// TIA Portal V20 export
TYPE "UDT_MTP_BinVlv"
TITLE = MTPDataObjectSUCLibrary/DataAssembly/BinVlv
   STRUCT
      CloseOp : Bool := FALSE;   // Close command from Operator (relevant, if StateOpAct) 0-->1:request from POL 1-->0 acknowledge from PEA(see Handshake)
      OpenOp : Bool := FALSE;   // Open command from Operator (relevant, if StateOpAct) 0-->1:request from POL 1-->0 acknowledge from PEA(see Handshake)
      OSLevel : Byte := 16#00;   // OSLevel variable
      StateChannel { ExternalWritable := 'False'} : Bool;   // Selection of the active Operation Mode interaction channel 0: the operator switches (*Op) shall be used 1: the automatic switches (*Aut) shall be used
      StateOffAut { ExternalWritable := 'False'} : Bool;   // Set OperationMode to Offline by automatic interaction (relevant, if StateChannel) 1:OperationMode is set to Offline 0:no operation
      StateOffOp : Bool;   // Set OperationMode to Offline by operator interaction (relevant, if not StateChannel) 0-->1:request to set OperationMode to Offline 1-->0:acknowledge by PEA
      StateOpAut { ExternalWritable := 'False'} : Bool;   // Set OperationMode to Operator by automatic interaction (relevant, if StateChannel) 1:OperationMode is set to Manual 0:no operation
      StateOpOp : Bool;   // Set OperationMode to Operator by operator interaction (relevant, if not StateChannel) 0-->1:request to set OperationMode to Manual 1-->0:acknowledge by PEA
      StateAutAut { ExternalWritable := 'False'} : Bool;   // Set OperationMode to Automatic by automatic interaction (relevant, if StateChannel) 1:OperationMode is set to Automatic 0:no operation
      StateAutOp : Bool;   // Set OperationMode to Automatic by operator interaction (relevant, if not StateChannel) 0-->1:request to set OperationMode is to Automatic 1-->0:acknowledge by PEA
      StateOpAct { ExternalWritable := 'False'} : Bool;   // 1: current mode is Operator 0: current mode is not Operator
      StateAutAct { ExternalWritable := 'False'} : Bool;   // 1: current mode is Automatic 0: current mode is not Automatic
      StateOffAct { ExternalWritable := 'False'} : Bool;   // 1: current mode is Offline 0: current mode is not Offline
      CSF { ExternalWritable := 'False'} : Bool;   // Reserved
      WQC { ExternalWritable := 'False'} : Byte := 16#FF;   // Worst Quality code
      CloseAut { ExternalWritable := 'False'} : Bool := FALSE;   // Set Valve to Close by Automatic (relevant, if StateAutAct) 1:close request 0:no close request
      OpenAut { ExternalWritable := 'False'} : Bool := FALSE;   // Set Valve to Open by Automatic (relevant, if StateAutAct) 1:open request 0:no open request
      Ctrl { ExternalWritable := 'False'} : Bool := FALSE;   // Valve Control 1:desired position is open 0:desired position is closed
      OpenFbkCalc { ExternalWritable := 'False'} : Bool := FALSE;   // Open Feedback Source 1: Calculated 0: Sensor detection
      CloseFbkCalc { ExternalWritable := 'False'} : Bool := FALSE;   // Close Feedback Source 1: Calculated 0: Sensor detection
      OpenFbk { ExternalWritable := 'False'} : Bool := FALSE;   // Open Feedback Signal 1:open 0:is not opened
      CloseFbk { ExternalWritable := 'False'} : Bool := FALSE;   // Close Feedback Signal 1:close 0:is not closed
      SafePos { ExternalWritable := 'False'} : Bool := FALSE;   // Safe Position 1: open 0: close
      SafePosEn { ExternalWritable := 'False'} : Bool;   // Hardware Safe Position enabled 1: Device has a safe position 0: Device has no safe position
      SafePosAct { ExternalWritable := 'False'} : Bool;   // Safe Position activated 1: Safe Position is activated (safe operation) 0: Safe Position is not activated (normal operation)
      PermEn { ExternalWritable := 'False'} : Bool := FALSE;   // Enables the Permission Lock 1:enabled 0:disabled
      Permit { ExternalWritable := 'False'} : Bool := FALSE;   // Permit allows control 1:permission is given 0:permission is not given
      IntlEn { ExternalWritable := 'False'} : Bool := FALSE;   // Enables the Interlock Lock 1:enabled 0:disabled
      Interlock { ExternalWritable := 'False'} : Bool := FALSE;   // Interlock prevents from being activated and sets it to safe position 1:interlock is not active 0:interlocking is active
      ProtEn { ExternalWritable := 'False'} : Bool := FALSE;   // Enables the Protection Lock 1:enabled 0:disabled
      Protect { ExternalWritable := 'False'} : Bool := FALSE;   // Protect prevents from being activated and sets it to safe position, requires a reset command 1: protect is not active 0: protect is active, requires reset
      ResetOp : Bool := FALSE;   // Reset from Operator (see Handshake) 0-->1:request from POL 1-->0: acknowledge from PEA
      ResetAut { ExternalWritable := 'False'} : Bool;   // Reset from Automatic 1:Reset executed 0:no Operation
   END_STRUCT;
END_TYPE
